ABB RAPID module: MainL.mod

MODULE MainL


PERS robtarget CupGrid{8} :=
[
    [[500, 425, 50],[0.707,0,0.707,0],[0,0,0,0],[0,9E+9,9E+9,9E+9,9E+9,9E+9]],
    [[500, 475, 50],[0.707,0,0.707,0],[0,0,0,0],[0,9E+9,9E+9,9E+9,9E+9,9E+9]],
    [[500, 525, 50],[0.707,0,0.707,0],[0,0,0,0],[0,9E+9,9E+9,9E+9,9E+9,9E+9]],
    [[500, 575, 50],[0.707,0,0.707,0],[0,0,0,0],[0,9E+9,9E+9,9E+9,9E+9,9E+9]],

    [[550, 425, 50],[0.707,0,0.707,0],[0,0,0,0],[0,9E+9,9E+9,9E+9,9E+9,9E+9]],
    [[550, 475, 50],[0.707,0,0.707,0],[0,0,0,0],[0,9E+9,9E+9,9E+9,9E+9,9E+9]],
    [[550, 525, 50],[0.707,0,0.707,0],[0,0,0,0],[0,9E+9,9E+9,9E+9,9E+9,9E+9]],
    [[550, 575, 50],[0.707,0,0.707,0],[0,0,0,0],[0,9E+9,9E+9,9E+9,9E+9,9E+9]]
];





PERS bool CupGridFull{8} := [FALSE,FALSE,FALSE,FALSE,FALSE,FALSE,FALSE,FALSE];

VAR num i;


    PROC main()
        ConfJ \Off;
        ConfL \Off;





    ENDPROC

ENDMODULE
